FUNCTION_BLOCK MockCoordinator IMPLEMENTS TcoCore.ITcoCoordinator
VAR
    _state : INT;
END_VAR

METHOD MoveNext : BOOL
_state := _state + 1;
END_METHOD

METHOD Retry : BOOL
VAR_INPUT
    inFromState : INT;
END_VAR
_state := inFromState;
END_METHOD

METHOD Terminate : BOOL
_state := 8005;
END_METHOD

END_FUNCTION_BLOCK

(* stored: Version 1.1.0.1, ProductVersion 3.1.4024.9
   POU MockCoordinator: Id {19596c80-18d9-089a-0b5b-3393ffeb1f11}, SpecialFunc None
   Method MoveNext: Id {44166f8a-8614-0309-3e0c-75242e506fe1}
   Method Retry: Id {6fbc6b6e-4c7f-004b-06ff-d3ee62e52a24}
   Method Terminate: Id {1dc80674-a43d-0e17-16c2-90bfdbe85e81} *)
